// TIA Portal V17 export
// export: Created 2024-03-30T11:14:47.6018442Z, ExportSetting WithDefaults, DisplayName Totally Integrated Automation Portal, DisplayVersion V17, DisplayName TIA Portal Openness, DisplayVersion V17, DisplayName TIA Portal Version Control Interface, DisplayVersion V17, DisplayName STEP 7 Professional, DisplayVersion V17, DisplayName STEP 7 Safety, DisplayVersion V17, DisplayName WinCC Advanced, DisplayVersion V17
DATA_BLOCK "PRG_VGR_Set_Positioning_DB"   // DB34
AUTHOR : A.Schaefer
VERSION : 0.1
// stored: AutoNumber true, DBAccessibleFromOPCUA true, DBAccessibleFromWebserver true, InstanceOfName PRG_VGR_Set_Positioning, InstanceOfType FB
"PRG_VGR_Set_Positioning"
   // VAR
   //    lx_Init { ExternalAccessible := 'False'; ExternalVisible := 'False'; ExternalWritable := 'False'} : Bool;
   //    lx_Start_TON_Wait { ExternalAccessible := 'False'; ExternalVisible := 'False'; ExternalWritable := 'False'} : Bool;
   //    lx_Start_Positioning_m { ExternalAccessible := 'False'; ExternalVisible := 'False'; ExternalWritable := 'False'} : Bool;
   //    lx_Start_FinalPositioning_m { ExternalAccessible := 'False'; ExternalVisible := 'False'; ExternalWritable := 'False'} : Bool;
   //    lx_Start_TON_State { ExternalAccessible := 'False'; ExternalVisible := 'False'; ExternalWritable := 'False'} : Bool;
   //    lt_TON_Wait { ExternalAccessible := 'False'; ExternalVisible := 'False'; ExternalWritable := 'False'} : Time;
   //    ldt_MQTT { ExternalAccessible := 'False'; ExternalVisible := 'False'; ExternalWritable := 'False'} : Date_And_Time;
   //    li_Return_LDT { ExternalAccessible := 'False'; ExternalVisible := 'False'; ExternalWritable := 'False'} : Int;
   //    li_Lights { ExternalAccessible := 'False'; ExternalVisible := 'False'; ExternalWritable := 'False'} : Int;
   //    li_Lights_old { ExternalAccessible := 'False'; ExternalVisible := 'False'; ExternalWritable := 'False'} : Int;
   //    lx_State_activ { ExternalAccessible := 'False'; ExternalVisible := 'False'; ExternalWritable := 'False'} : Bool;
   //    li_StepCase { ExternalAccessible := 'False'; ExternalVisible := 'False'; ExternalWritable := 'False'} : Int;
   //    li_Counter { ExternalAccessible := 'False'; ExternalVisible := 'False'; ExternalWritable := 'False'} : Int;
   //    ldi_Pos_SLD_X { ExternalAccessible := 'False'; ExternalVisible := 'False'; ExternalWritable := 'False'} : DInt;
   //    ldi_Pos_SLD_Y { ExternalAccessible := 'False'; ExternalVisible := 'False'; ExternalWritable := 'False'} : DInt;
   //    ldi_Pos_SLD_Z { ExternalAccessible := 'False'; ExternalVisible := 'False'; ExternalWritable := 'False'} : DInt;
   //    ldi_Pos_Horizontal { ExternalAccessible := 'False'; ExternalVisible := 'False'; ExternalWritable := 'False'} : DInt;
   //    ldi_Pos_Vertical { ExternalAccessible := 'False'; ExternalVisible := 'False'; ExternalWritable := 'False'} : DInt;
   //    ldi_Pos_Rotate { ExternalAccessible := 'False'; ExternalVisible := 'False'; ExternalWritable := 'False'} : DInt;
   //    ldi_Offset_Vertical { ExternalAccessible := 'False'; ExternalVisible := 'False'; ExternalWritable := 'False'} : DInt;
   //    ls_Color { ExternalAccessible := 'False'; ExternalVisible := 'False'; ExternalWritable := 'False'} : String;
   //    ls_Target { ExternalAccessible := 'False'; ExternalVisible := 'False'; ExternalWritable := 'False'} : String;
   //    lfb_TON_Wait { ExternalAccessible := 'False'; ExternalVisible := 'False'; ExternalWritable := 'False'} : TON_TIME;
   //    lfb_TON_State { ExternalAccessible := 'False'; ExternalVisible := 'False'; ExternalWritable := 'False'} : TON_TIME;
   //    lfb_R_Trig_Deaktivate { ExternalAccessible := 'False'; ExternalVisible := 'False'; ExternalWritable := 'False'} : R_TRIG;
   //    lfb_R_Trig_NiO { ExternalAccessible := 'False'; ExternalVisible := 'False'; ExternalWritable := 'False'} : R_TRIG;
   // END_VAR
BEGIN
END_DATA_BLOCK
